// Mitsubishi GX Works2 project: kremboDay   PLC: FX3G

// global labels: Global1
VAR_GLOBAL
  StartSwitch AT X007 : BOOL;
END_VAR
VAR_GLOBAL CONSTANT
  MinimunCream : INT := 300;
END_VAR
VAR_GLOBAL
  InitialCream AT D1100 : REAL;
  EnoughCream AT M1 : BOOL;
END_VAR
VAR_GLOBAL CONSTANT
  MinimumChoc : INT := 240;
END_VAR
VAR_GLOBAL
  InitialChoc AT D1102 : REAL;
  EnoughChoc AT M2 : BOOL;
  InitialBisq AT D1104 : REAL;
END_VAR
VAR_GLOBAL CONSTANT
  MinimumBisq : INT;
END_VAR
VAR_GLOBAL
  EnoughBisq AT M3 : BOOL;
  InitialDay AT M70 : BOOL;
  CreamContainer AT D1106 : REAL;
  ChocContainer AT D1108 : REAL;
  BisqContainer AT D1110 : REAL;
  DayStarted AT M54 : BOOL;
  finale AT M11 : BOOL;
  temp AT M22 : BOOL;
  blink AT M6 : BOOL;
  workingDay AT Y007 : BOOL;
  EndPacking AT M90 : BOOL;
  StartTopping AT X011 : BOOL;
  SwitchToppingMach AT X010 : BOOL;
  SystemOn AT M0 : BOOL;
  CameraSignal AT X003 : BOOL;
  Error AT X005 : BOOL;
  PlateFit AT X001 : BOOL;
  Sen_15 AT X004 : BOOL;
  ToppingOn AT Y004 : BOOL;
  Sen_30 AT X006 : BOOL;
END_VAR
VAR_GLOBAL CONSTANT
  CreamBatch : REAL := 300;
END_VAR
VAR_GLOBAL
  ToppingContainer AT D1110 : INT;
  TransCream AT M80 : BOOL;
  Transfer AT M12 : BOOL;
  CommitTransfer AT CS0 : BOOL;
END_VAR
VAR_GLOBAL CONSTANT
  Time40 : REAL;
END_VAR
VAR_GLOBAL
  TC1 AT TC1 : BOOL;
  TC1 AT TC1 : BOOL;
  TC1 AT TC1 : BOOL;
  TC1 AT TC1 : BOOL;
  TC1 AT TC1 : BOOL;
  TC1 AT TC1 : BOOL;
  TC1 AT TC1 : BOOL;
  TC1 AT TC1 : BOOL;
  tc2 AT TC2 : BOOL;
  TC1 AT TC1 : BOOL;
  CONTER AT TC1 : BOOL;
  StopBlink AT TS1 : BOOL;
  StartBlink AT M33 : BOOL;
  ts3 AT TS3 : BOOL;
  TS3 AT TS3 : BOOL;
  TS3 AT TS3 : BOOL;
  TS3 AT TS3 : BOOL;
  TS3 AT TS3 : BOOL;
  TS3 AT TS3 : BOOL;
  TS3 AT TS3 : BOOL;
  TS3 AT TS3 : BOOL;
  Fic1 AT M20 : BOOL;
  ts2 AT TS2 : BOOL;
  TS3 AT TS3 : BOOL;
  TransLed2 AT Y001 : BOOL;
  Time4 AT D1112 : INT;
  tc3 AT TC3 : BOOL;
  TransLed1 AT Y000 : BOOL;
  TC2 AT TC2 : BOOL;
  FinalBlink AT TS6 : BOOL;
  CounterFinished AT CS1 : BOOL;
  CounterFinished1 AT CS1 : BOOL;
END_VAR
VAR_GLOBAL CONSTANT
  SixMin : REAL := 6;
  gr300 : REAL := 300;
  unit6 : REAL := 300;
END_VAR
VAR_GLOBAL
  EnoughStock AT M100 : BOOL;
  TransBeforeSprink AT X011 : BOOL;
END_VAR
VAR_GLOBAL CONSTANT
  BisqBatch : REAL := 6;
END_VAR
VAR_GLOBAL
  SprinkContainer AT D1114 : INT;
  BisqBox AT D1116 : REAL;
  TempUnder15 AT X004 : BOOL;
  SprinkOn AT Y004 : BOOL;
  TempUnder30 AT X011 : BOOL;
  TempOver30 AT X002 : BOOL;
  SwitchSprinkMach AT X010 : BOOL;
  StartSprinkMach AT M0 : BOOL;
  TransBisq AT M81 : BOOL;
  TransKrembo AT M12 : BOOL;
  StartCoat AT X006 : BOOL;
  AnalogInput1 AT D8280 : INT;
  ChoclateInput AT D1118 : REAL;
END_VAR
VAR_GLOBAL CONSTANT
  NormalRange : REAL := 400;
END_VAR
VAR_GLOBAL
  NormalizedInput AT M13 : BOOL;
END_VAR
VAR_GLOBAL CONSTANT
  Six : REAL := 6;
  Five : REAL;
  SingleCoat : REAL := 120;
  DoubleCoat : REAL := 240;
END_VAR
VAR_GLOBAL
  CoatingContainer AT D1120 : REAL;
  ChocContainerReady AT M16 : BOOL;
  CoatingTime AT TC4 : BOOL;
  CoatingInProcess AT Y003 : BOOL;
END_VAR

// task Task_01 (event TRUE, interval 0, priority 31): POU_01

PROGRAM POU_01
VAR CONSTANT
  gr240 : REAL := 240;
  Five : REAL := 5;
  FiveSeconds : REAL := 5;
END_VAR
(* structured ladder/FBD written out as ST: instructions are called as NAME(EN, inputs, outputs); _pN, _eN, _tN stand for wires *)
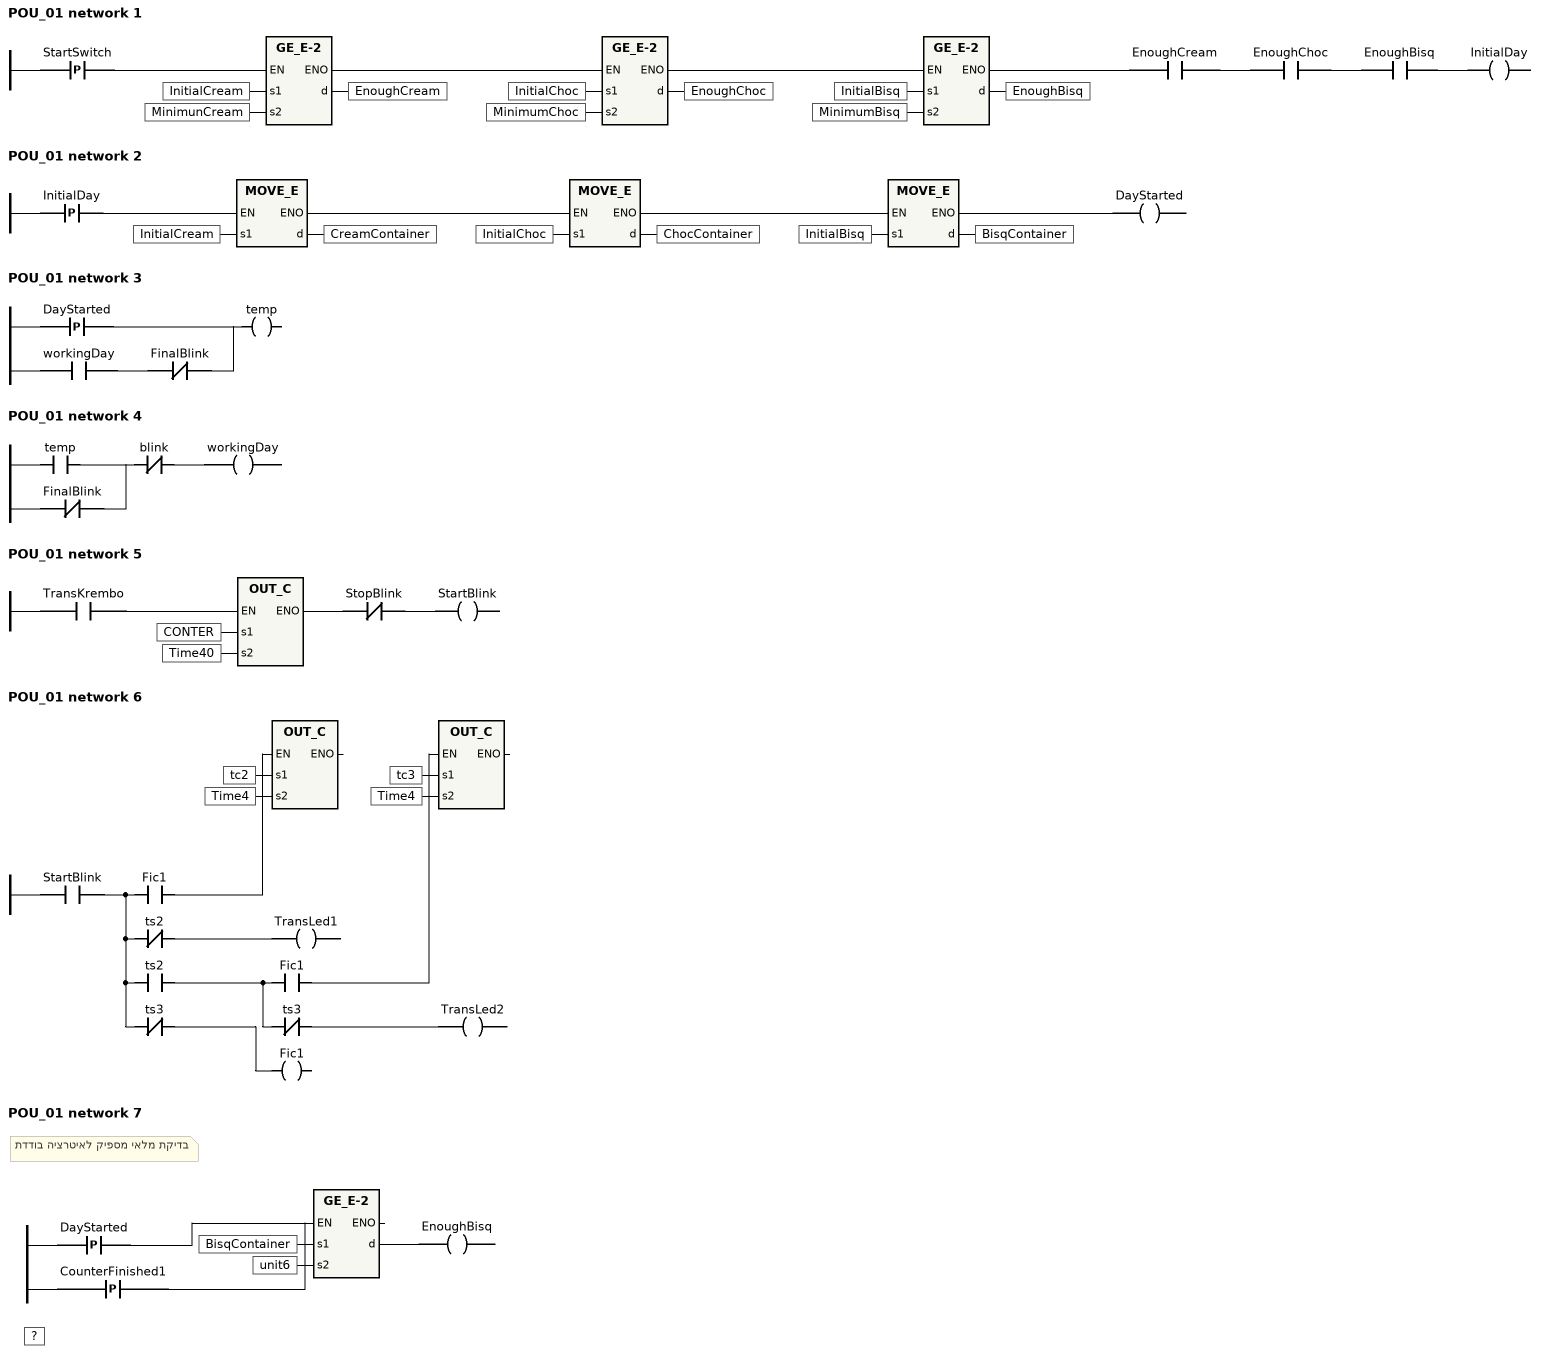
(* network 1 *)
_e1 := GE_E(LDP(TRUE, StartSwitch), InitialCream, MinimunCream, EnoughCream);
_e2 := GE_E(_e1, InitialChoc, MinimumChoc, EnoughChoc);
_e3 := GE_E(_e2, InitialBisq, MinimumBisq, EnoughBisq);
InitialDay := _e3 AND EnoughCream AND EnoughChoc AND EnoughBisq;
(* network 2 *)
_e1 := MOVE_E(LDP(TRUE, InitialDay), InitialCream, CreamContainer);
_e2 := MOVE_E(_e1, InitialChoc, ChocContainer);
_e3 := MOVE_E(_e2, InitialBisq, BisqContainer);
DayStarted := _e3;
(* network 3 *)
temp := LDP(TRUE, DayStarted) OR (workingDay AND NOT FinalBlink);
(* network 4 *)
workingDay := (temp OR (NOT FinalBlink)) AND NOT blink;
(* network 5 *)
_e1 := OUT_C(TransKrembo, CONTER, Time40);
StartBlink := _e1 AND NOT StopBlink;
(* network 6 *)
OUT_C(StartBlink AND Fic1, tc2, Time4);
TransLed1 := StartBlink AND NOT ts2;
_p1 := StartBlink AND ts2;
OUT_C(_p1 AND Fic1, tc3, Time4);
TransLed2 := _p1 AND NOT ts3;
Fic1 := StartBlink AND NOT ts3;
(* network 7 *)
(* בדיקת מלאי מספיק לאיטרציה בודדת *)
GE_E(LDP(TRUE, DayStarted) OR LDP(TRUE, CounterFinished1), BisqContainer, unit6, _t1);
EnoughBisq := _t1;
(* not connected to any output: ? *)
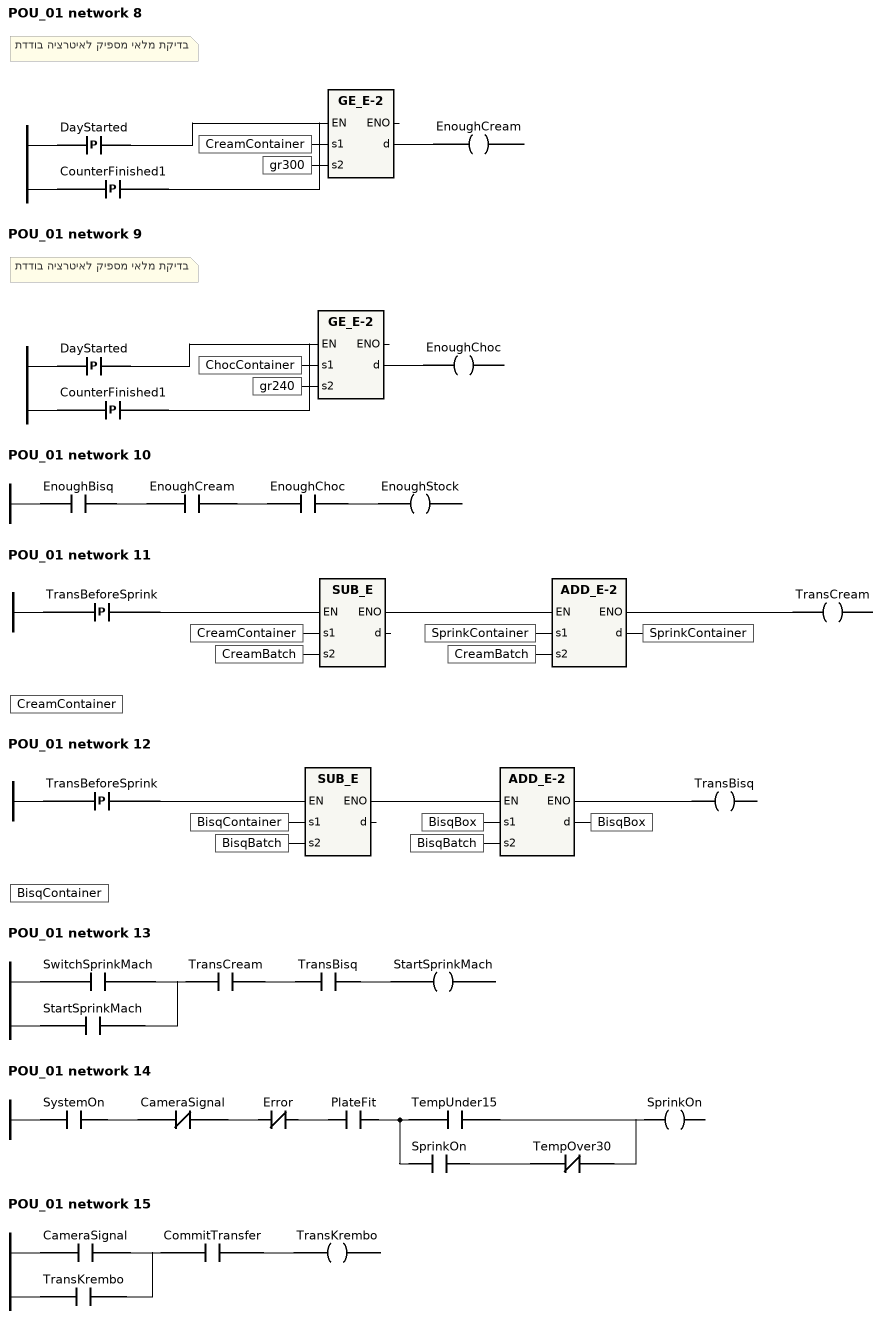
(* network 8 *)
(* בדיקת מלאי מספיק לאיטרציה בודדת *)
GE_E(LDP(TRUE, DayStarted) OR LDP(TRUE, CounterFinished1), CreamContainer, gr300, _t1);
EnoughCream := _t1;
(* network 9 *)
(* בדיקת מלאי מספיק לאיטרציה בודדת *)
GE_E(LDP(TRUE, DayStarted) OR LDP(TRUE, CounterFinished1), ChocContainer, gr240, _t1);
EnoughChoc := _t1;
(* network 10 *)
EnoughStock := EnoughBisq AND EnoughCream AND EnoughChoc;
(* network 11 *)
_e1 := SUB_E(LDP(TRUE, TransBeforeSprink), CreamContainer, CreamBatch, _open);
_e2 := ADD_E(_e1, SprinkContainer, CreamBatch, SprinkContainer);
TransCream := _e2;
CreamContainer := (* unconnected *);
(* network 12 *)
_e1 := SUB_E(LDP(TRUE, TransBeforeSprink), BisqContainer, BisqBatch, _open);
_e2 := ADD_E(_e1, BisqBox, BisqBatch, BisqBox);
TransBisq := _e2;
BisqContainer := (* unconnected *);
(* network 13 *)
StartSprinkMach := ((SwitchSprinkMach OR StartSprinkMach) AND TransCream) AND TransBisq;
(* network 14 *)
_p1 := SystemOn AND NOT CameraSignal AND NOT Error AND PlateFit;
SprinkOn := (_p1 AND TempUnder15) OR (_p1 AND SprinkOn AND NOT TempOver30);
(* network 15 *)
TransKrembo := (CameraSignal OR TransKrembo) AND CommitTransfer;
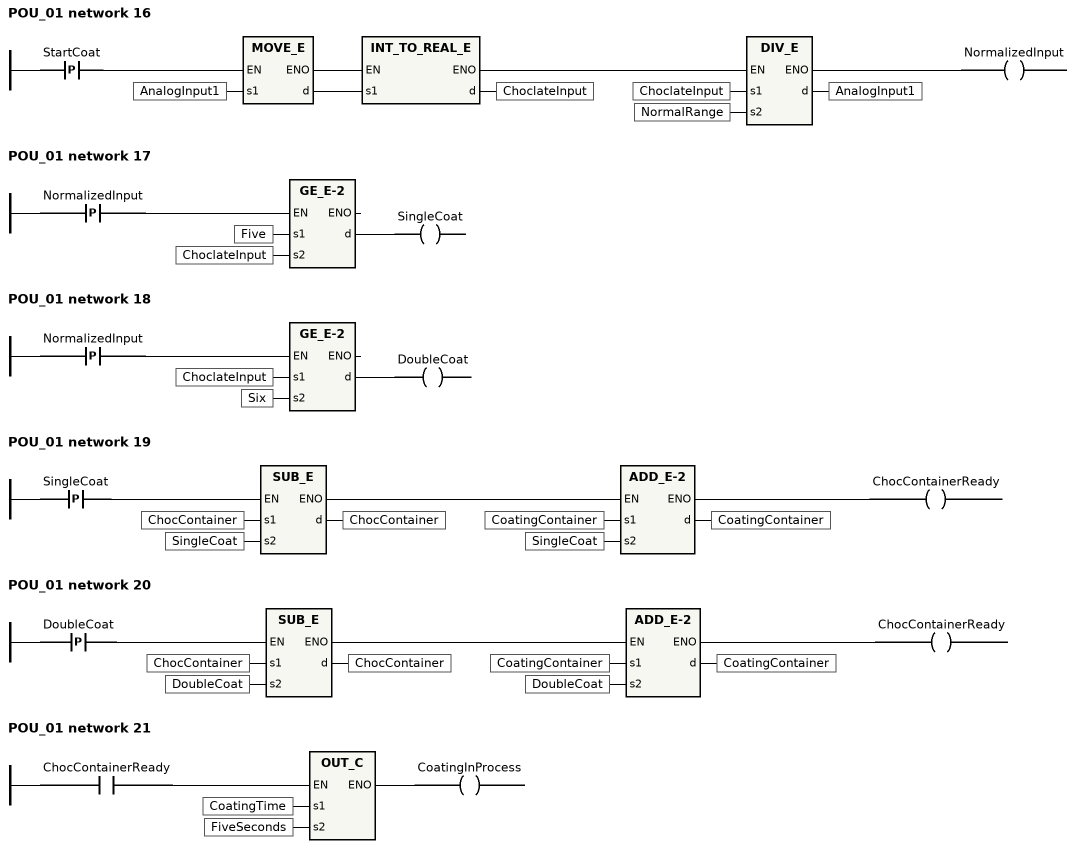
(* network 16 *)
_e2 := MOVE_E(LDP(TRUE, StartCoat), AnalogInput1, _t1);
_e3 := INT_TO_REAL_E(_e2, _t1, ChoclateInput);
_e4 := DIV_E(_e3, ChoclateInput, NormalRange, AnalogInput1);
NormalizedInput := _e4;
(* network 17 *)
GE_E(LDP(TRUE, NormalizedInput), Five, ChoclateInput, _t1);
SingleCoat := _t1;
(* network 18 *)
GE_E(LDP(TRUE, NormalizedInput), ChoclateInput, Six, _t1);
DoubleCoat := _t1;
(* network 19 *)
_e1 := SUB_E(LDP(TRUE, SingleCoat), ChocContainer, SingleCoat, ChocContainer);
_e2 := ADD_E(_e1, CoatingContainer, SingleCoat, CoatingContainer);
ChocContainerReady := _e2;
(* network 20 *)
_e1 := SUB_E(LDP(TRUE, DoubleCoat), ChocContainer, DoubleCoat, ChocContainer);
_e2 := ADD_E(_e1, CoatingContainer, DoubleCoat, CoatingContainer);
ChocContainerReady := _e2;
(* network 21 *)
_e1 := OUT_C(ChocContainerReady, CoatingTime, FiveSeconds);
CoatingInProcess := _e1;
END_PROGRAM
